// TIA Portal V21 export
TYPE "LBC_typeDigitalSignalInterface"
TITLE = LBC_typeDigitalSignalInterface
// Module interface for external systems
   STRUCT
      commands : "LBC_typeInterfaceCommands";
      monitoring { ExternalWritable := 'False'} : "LBC_typeDigitalSignalProcessValues";
      configuration : "LBC_typeDigitalSignalConfiguration";
   END_STRUCT;
END_TYPE
